INTERFACE I_DatatypeAddedEvent EXTENDS I_Event

PROPERTY PUBLIC Target : I_Datatype
GET
END_GET
END_PROPERTY

END_INTERFACE

(* stored: Version 1.1.0.1, ProductVersion 3.1.4024.12
   Itf I_DatatypeAddedEvent: Id {ce71c747-2365-0ade-1a33-35557bb6d2ea}
   Property Target: Id {c6c7f274-3c0d-033d-131c-3dd58a0b6e43}
   Get Get: Id {d830ac5f-1b6b-0325-1667-5377a1efef1f} *)
